KUKA KRL program: testprog.src

&ACCESS RVP
&REL 22
&PARAM TEMPLATE = C:\KRC\Roboter\Template\ExpertVorgabe
&PARAM EDITMASK = *
DEF TestProg( )

;--------- Declarations ------------------------------------
EXT BAS (BAS_COMMAND :IN,REAL :IN )

;---------- Init -------------------------------------------
BAS (#INITMOV,0 ) ;Initialicing the defaults for Vel and so on

; SAK
PTP {AXIS: A1 0,A2 -90,A3 90,A4 0,A5 0,A6 0}

; Velocity for LIN points
$VEL.CP = 2 ; m/s



END
